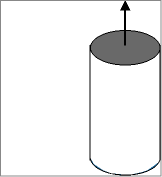
VISUALIZATION VISU_Tube_Top_9  // 162x177
VAR_IN_OUT
	azi : LREAL;
END_VAR
    Ellipse (90,140 70x35)
        p2858320360: azi
    Polygon (90,45) (160,45) (160,157) (158,162) (154,165) (147,170) (141,172) (132,174) (121,174) (111,173) (103,170) (94,164) (90,157)
        p2858320360: azi
    Ellipse (90,30 70x35)
        p2858320360: azi
    Polygon (120,10) (125,0) (130,10)
        p2858320360: azi
    Polyline (125,45) (125,10)
        p2858320360: azi
    Polyline (160,160) (160,45)
        p2858320360: azi
    Polyline (90,160) (90,45)
        p2858320360: azi
END_VISUALIZATION

(* stored: Version 1.1.0.1, ProductVersion 3.1.4018.5
   Visu VISU_Tube_Top_9: Id {13a5717c-806c-4152-95be-cd937079e0bb} *)
